Staubli VAL3: SetFrame.pgx

public program SetFrame(string x_sFrame)
begin
  //
  sFrameName=x_sFrame
end
